(* PLC project BoxTurtle_Control, BoxTurtle FilamentFeeder 1.0 *)
(* stored: creationDateTime 2025-11-21T12:00:00, modificationDateTime 2025-11-21T12:00:00 *)

TYPE E_FeederState : (IDLE := 0, CUTTING := 10, UNLOADING := 20, LOADING := 30, ERROR := 99);
END_TYPE

FUNCTION_BLOCK FB_Cutter
  VAR_INPUT
    bExecute : BOOL;
  END_VAR
  VAR_OUTPUT
    bDone : BOOL;
    bServoSignal : BOOL;
  END_VAR
  VAR
    iStep : INT := 0;
    fbTimer : TON;
  END_VAR

            
              
CASE iStep OF
  0: (* Idle *)
    bDone := FALSE;
    bServoSignal := FALSE;
    IF bExecute THEN
      iStep := 10;
    END_IF;

  10: (* Actuate Servo *)
    bServoSignal := TRUE;
    fbTimer(IN:=TRUE, PT:=T#500MS);
    IF fbTimer.Q THEN
      fbTimer(IN:=FALSE);
      iStep := 20;
    END_IF;

  20: (* Retract Servo *)
    bServoSignal := FALSE;
    fbTimer(IN:=TRUE, PT:=T#500MS);
    IF fbTimer.Q THEN
      fbTimer(IN:=FALSE);
      bDone := TRUE;
      iStep := 30;
    END_IF;

  30: (* Wait for Reset *)
    IF NOT bExecute THEN
      bDone := FALSE;
      iStep := 0;
    END_IF;
END_CASE;
              
            
          
END_FUNCTION_BLOCK

FUNCTION_BLOCK FB_Lane
  VAR_INPUT
    bLoad : BOOL;
    bUnload : BOOL;
    bFilamentSensor : BOOL;
  END_VAR
  VAR_OUTPUT
    bMotorRun : BOOL;
    bMotorDir : BOOL;
    bBusy : BOOL;
    bDone : BOOL;
  END_VAR
  VAR
    iState : INT;
  END_VAR

            
              
CASE iState OF
  0: (* Idle *)
    bMotorRun := FALSE;
    bBusy := FALSE;
    bDone := FALSE;
    IF bLoad THEN
      iState := 10;
    ELSIF bUnload THEN
      iState := 20;
    END_IF;

  10: (* Loading *)
    bBusy := TRUE;
    bMotorDir := TRUE;
    bMotorRun := TRUE;
    (* Run until sensor sees filament *)
    IF bFilamentSensor THEN
      bMotorRun := FALSE;
      bDone := TRUE;
      iState := 30;
    END_IF;

  20: (* Unloading *)
    bBusy := TRUE;
    bMotorDir := FALSE;
    bMotorRun := TRUE;
    (* Run until sensor loses filament *)
    IF NOT bFilamentSensor THEN
      bMotorRun := FALSE;
      bDone := TRUE;
      iState := 30;
    END_IF;

  30: (* Wait for Command Clear *)
    IF NOT bLoad AND NOT bUnload THEN
      bDone := FALSE;
      bBusy := FALSE;
      iState := 0;
    END_IF;
END_CASE;
              
            
          
END_FUNCTION_BLOCK

PROGRAM PRG_Main
  VAR_INPUT
    iRequestedTool : INT;
    bStartChange : BOOL;
    Inputs_Sensors : ARRAY[1..4] OF BOOL;
  END_VAR
  VAR_OUTPUT
    Outputs_MotorRun : ARRAY[1..4] OF BOOL;
    Outputs_MotorDir : ARRAY[1..4] OF BOOL;
    Output_CutterServo : BOOL;
    bSystemReady : BOOL;
  END_VAR
  VAR
    eState : E_FeederState := IDLE;
    iCurrentTool : INT := 0;
    fbLanes : ARRAY[1..4] OF FB_Lane;
    fbCutter : FB_Cutter;
    i : INT;
  END_VAR

            
              
(* Main State Machine *)
CASE eState OF
  E_FeederState.IDLE:
    bSystemReady := TRUE;
    IF bStartChange AND (iRequestedTool <> iCurrentTool) THEN
      bSystemReady := FALSE;
      eState := E_FeederState.CUTTING;
    END_IF;

  E_FeederState.CUTTING:
    (* Step 1: Cut the current filament if any is loaded *)
    IF iCurrentTool > 0 THEN
      fbCutter(bExecute := TRUE);
      IF fbCutter.bDone THEN
        fbCutter(bExecute := FALSE);
        eState := E_FeederState.UNLOADING;
      END_IF;
    ELSE
      (* No tool loaded, skip cut/unload *)
      eState := E_FeederState.LOADING;
    END_IF;

  E_FeederState.UNLOADING:
    (* Step 2: Unload the old tool *)
    fbLanes[iCurrentTool](bUnload := TRUE, bFilamentSensor := Inputs_Sensors[iCurrentTool]);
    
    Outputs_MotorRun[iCurrentTool] := fbLanes[iCurrentTool].bMotorRun;
    Outputs_MotorDir[iCurrentTool] := fbLanes[iCurrentTool].bMotorDir;

    IF fbLanes[iCurrentTool].bDone THEN
      fbLanes[iCurrentTool](bUnload := FALSE); (* Reset Lane *)
      iCurrentTool := 0; (* Cleared *)
      eState := E_FeederState.LOADING;
    END_IF;

  E_FeederState.LOADING:
    (* Step 3: Load the new tool *)
    fbLanes[iRequestedTool](bLoad := TRUE, bFilamentSensor := Inputs_Sensors[iRequestedTool]);

    Outputs_MotorRun[iRequestedTool] := fbLanes[iRequestedTool].bMotorRun;
    Outputs_MotorDir[iRequestedTool] := fbLanes[iRequestedTool].bMotorDir;

    IF fbLanes[iRequestedTool].bDone THEN
      fbLanes[iRequestedTool](bLoad := FALSE); (* Reset Lane *)
      iCurrentTool := iRequestedTool;
      eState := E_FeederState.IDLE;
    END_IF;

  E_FeederState.ERROR:
    (* Error handling logic here *)
    bSystemReady := FALSE;

END_CASE;

(* Map Cutter Output *)
Output_CutterServo := fbCutter.bServoSignal;
              
            
          
END_PROGRAM

CONFIGURATION Config0
  RESOURCE Res0 ON PLC
    TASK TaskMain(INTERVAL := T#10ms, PRIORITY := 0);
    PROGRAM InstMain WITH TaskMain : PRG_Main;
  END_RESOURCE
END_CONFIGURATION
